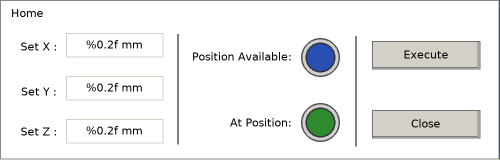
VISUALIZATION Home  // 500x160
    Rectangle (0,0 500x159)
    Label (-36,32 150x30), "Set X :"
    Label (-36,77 150x30), "Set Y :"
    Label (-36,117 150x30), "Set Z :"
    Textfield (66,33 97x24), "%0.2f mm", text variable: Set_Pos_XHome
        OnMouseDown: write Set_Pos_XHome via VisuDialogs.Numpad
    Textfield (66,76 97x24), "%0.2f mm", text variable: Set_Pos_YHome
        OnMouseClick: write Set_Pos_YHome via VisuDialogs.Numpad
    Textfield (66,119 97x24), "%0.2f mm", text variable: Set_Pos_ZHome
        OnMouseClick: write Set_Pos_ZHome via VisuDialogs.Numpad
    Line (192,47)
    Line (178,144) (178,34)
    Lamp1 (298,35 45x45), variable: Home.Pos_Exists, style: Lamp-Lamp1-Blue
    Label (167,42 150x30), "Position Available:"
    Line (192,109)
    Lamp1 (298,100 45x45), variable: out_b_inHome, style: Lamp-Lamp1-Green
    Label (206,107 110x32), "At Position:"
    Line (356,146) (356,36)
    Button (372,41 108x28), "Execute", invisible if: Home.Pos_NotValid
        toggle in_b_MoveHome
    Button (372,110 108x28), "Close"
        OnMouseClick: CloseDialog Dialog=Home, Result=OK, NumpadKeypadSet=True
    Rectangle (1,1 498x25), "Home"
END_VISUALIZATION

(* stored: Version 1.1.0.1, ProductVersion 3.1.4018.9
   Visu Home: Id {5263df9e-bc3c-4b9e-8201-38e61babd047} *)
